(* PLC project My Custom Library, OpenPLC My Custom Library 1.0, author Thiago Alves *)
(* stored: creationDateTime 2020-01-21T09:44:11, modificationDateTime 2020-01-21T09:44:11 *)

(* This block outputs the sum of input I0 and 10. *)
FUNCTION_BLOCK Test
  VAR_INPUT
    I0 : INT;  (* Insert an integer here *)
    ACTIVE : BOOL;  (* 0 – block does nothing, 1 – block sums 10 to integer in I0 *)
  END_VAR
  VAR_OUTPUT
    OUT : INT;  (* This is the output: I0 + 10 *)
  END_VAR

            IF ACTIVE = TRUE THEN
OUT := I0 + 10;
END_IF;
          
END_FUNCTION_BLOCK
